% RSLogix 500 project SIMPLE CONTROL LOGIC PRACTICE.RSS, saved by version 8.30.00.16 %
PROJECT "SIM_PLC"    % processor: Bul.1763 MicroLogix 1100 Series B %

PROGRAM FILES
  LAD 2 "MAIN"  4 rungs
  LAD 3 "INPUTS"  3 rungs
  LAD 4 "OUTPUTS"  3 rungs
  LAD 5 "CTRL LOGIC"  9 rungs

DATA FILES
  O0 OUTPUT  5 elements
  I1 INPUT  7 elements
  S2 STATUS  66 elements
  B3 BINARY  1 elements
  T4 TIMER  5 elements
  C5 COUNTER  1 elements
  R6 CONTROL  1 elements
  N7 INTEGER  2 elements
  F8 FLOAT  1 elements

LADDER 2 "MAIN"
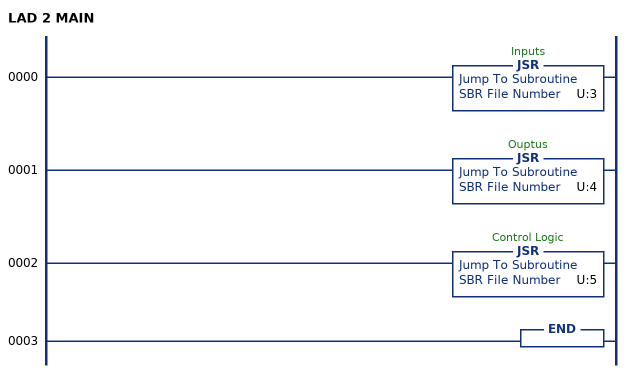
% Rung: 0 %
SOR JSR U:3 EOR
%   U:3  "Inputs" %
% Rung: 1 %
SOR JSR U:4 EOR
%   U:4  "Ouptus" %
% Rung: 2 %
SOR JSR U:5 EOR
%   U:5  "Control Logic" %
% Rung: 3 %
SOR END EOR

LADDER 3 "INPUTS"
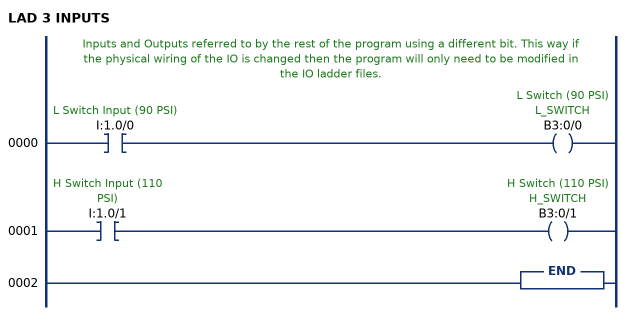
% Rung: 0 %
% Inputs and Outputs referred to by the rest of the program using a different bit. This way if the physical wiring of the IO is changed then the program will only need to be modified in the IO ladder files. %
SOR XIC I:1.0/0 OTE B3:0/0 EOR
%   I:1.0/0  "L Switch Input (90 PSI)" %
%   B3:0/0  L_SWITCH  "L Switch (90 PSI)" %
% Rung: 1 %
SOR XIC I:1.0/1 OTE B3:0/1 EOR
%   I:1.0/1  "H Switch Input (110 PSI)" %
%   B3:0/1  H_SWITCH  "H Switch (110 PSI)" %
% Rung: 2 %
SOR END EOR

LADDER 4 "OUTPUTS"
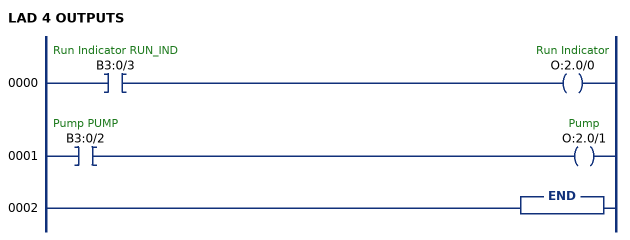
% Rung: 0 %
SOR XIC B3:0/3 OTE O:2.0/0 EOR
%   B3:0/3  RUN_IND  "Run Indicator" %
%   O:2.0/0  "Run Indicator" %
% Rung: 1 %
SOR XIC B3:0/2 OTE O:2.0/1 EOR
%   B3:0/2  PUMP  "Pump" %
%   O:2.0/1  "Pump" %
% Rung: 2 %
SOR END EOR

LADDER 5 "CTRL LOGIC"
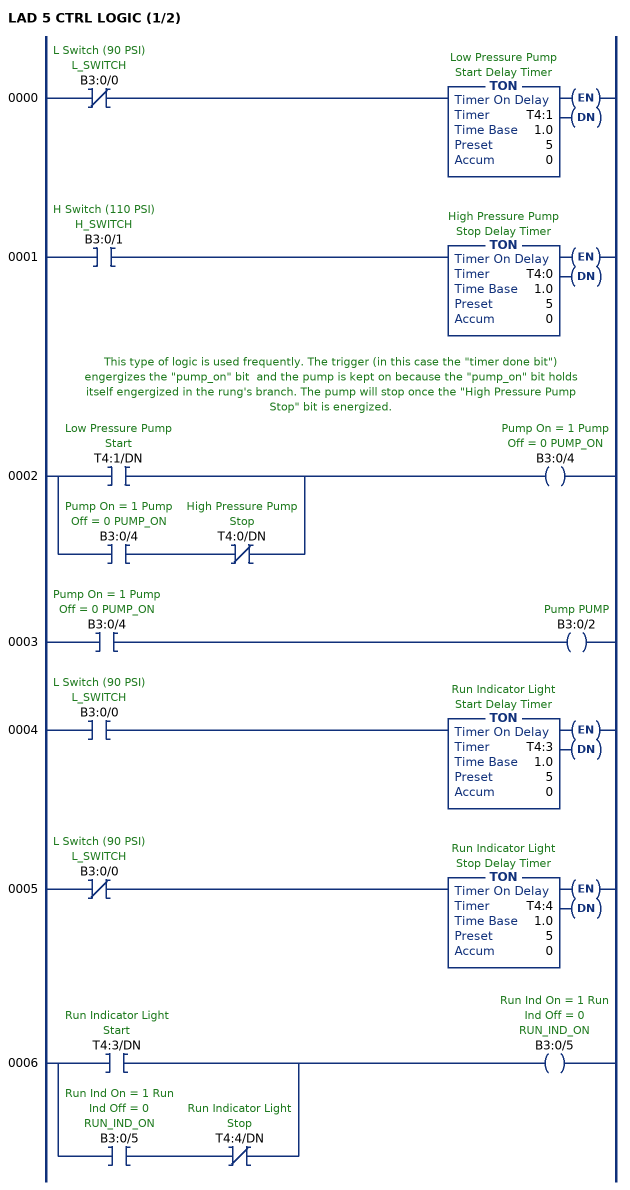
% Rung: 0 %
SOR XIO B3:0/0 TON T4:1 1.0 5 0 EOR
%   B3:0/0  L_SWITCH  "L Switch (90 PSI)" %
%   T4:1  "Low Pressure Pump Start Delay Timer" %
% Rung: 1 %
SOR XIC B3:0/1 TON T4:0 1.0 5 0 EOR
%   B3:0/1  H_SWITCH  "H Switch (110 PSI)" %
%   T4:0  "High Pressure Pump Stop Delay Timer" %
% Rung: 2 %
% This type of logic is used frequently. The trigger (in this case the "timer done bit") engergizes the "pump_on" bit  and the pump is kept on because the "pump_on" bit holds itself engergized in the rung's branch. The pump will stop once the "High Pressure Pump Stop" bit is energized. %
SOR BST XIC T4:1/DN NXB XIC B3:0/4 XIO T4:0/DN BND OTE B3:0/4 EOR
%   T4:1/DN  "Low Pressure Pump Start" %
%   B3:0/4  PUMP_ON  "Pump On = 1 Pump Off = 0" %
%   T4:0/DN  "High Pressure Pump Stop" %
% Rung: 3 %
SOR XIC B3:0/4 OTE B3:0/2 EOR
%   B3:0/4  PUMP_ON  "Pump On = 1 Pump Off = 0" %
%   B3:0/2  PUMP  "Pump" %
% Rung: 4 %
SOR XIC B3:0/0 TON T4:3 1.0 5 0 EOR
%   B3:0/0  L_SWITCH  "L Switch (90 PSI)" %
%   T4:3  "Run Indicator Light Start Delay Timer" %
% Rung: 5 %
SOR XIO B3:0/0 TON T4:4 1.0 5 0 EOR
%   B3:0/0  L_SWITCH  "L Switch (90 PSI)" %
%   T4:4  "Run Indicator Light Stop Delay Timer" %
% Rung: 6 %
SOR BST XIC T4:3/DN NXB XIC B3:0/5 XIO T4:4/DN BND OTE B3:0/5 EOR
%   T4:3/DN  "Run Indicator Light Start" %
%   B3:0/5  RUN_IND_ON  "Run Ind On = 1 Run Ind Off = 0" %
%   T4:4/DN  "Run Indicator Light Stop" %

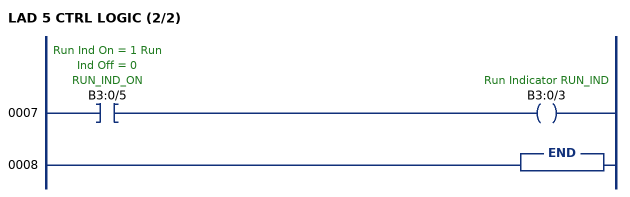
% Rung: 7 %
SOR XIC B3:0/5 OTE B3:0/3 EOR
%   B3:0/5  RUN_IND_ON  "Run Ind On = 1 Run Ind Off = 0" %
%   B3:0/3  RUN_IND  "Run Indicator" %
% Rung: 8 %
SOR END EOR

OTHER DOCUMENTED ADDRESSES
  I:3.0  "Pressure Switch Input"
  N7:0  "Pressure (0-110 PSI)"
  N7:1  "Pressure (0-100%)"

DATA TABLE (non-zero values as saved)
DATA T4
% .PRE .ACC %
% T4:0 % 5 0
% T4:1 % 5 0
% T4:3 % 5 0
% T4:4 % 5 0
